TYPE E_KMotorVFD_States : (
	KMOTORVFDSTATE_DISABLED,
	KMOTORVFDSTATE_ENABLING,
	KMOTORVFDSTATE_PU_TYPE_CHECK,
	KMOTORVFDSTATE_SERIAL_CHECK,
	KMOTORVFDSTATE_SERIAL_CU_CHECK,
	KMOTORVFDSTATE_FACTORY_RESET,
	KMOTORVFDSTATE_FACTORY_RESET_CHECK,
	KMOTORVFDSTATE_WAIT_FOR_ETHERCAT_RESET,
	KMOTORVFDSTATE_ETHERCAT_RESET,
	KMOTORVFDSTATE_ETHERCAT_RESET_CHECK,
	KMOTORVFDSTATE_PARAMETER_WRITE,
	KMOTORVFDSTATE_STOPPING,
	KMOTORVFDSTATE_STOPPED,
	KMOTORVFDSTATE_FWD,
	KMOTORVFDSTATE_REV,
	KMOTORVFDSTATE_JOG_MODE,
	KMOTORVFDSTATE_ERROR_DRIVE_FAULT
);
END_TYPE

(* stored: Version 1.1.0.1, ProductVersion 3.1.4024.12
   DUT E_KMotorVFD_States: Id {ba34b632-5ae6-4d8e-9d6b-76ac057d056a} *)
